{attribute addProperty BoxType "BK1250-0000-0019"}
{attribute addProperty Id "A_0001_KL_6211_ASI_Master_Parameter_Interface_and_6_Byte_11_ASI_Slaves_PowerKL6211_9210FF7200A_0002_KL_6211_ASI_Master_Parameter_Interface_and_6_Byte_11_ASI_Slaves_PowerKL_F309D72200A_0005_KL_6211_ASI_Master_Parameter_Interface_and_16_Byte_31_ASI_Slaves_PowerKL_54D8646000A_0006_KL_6211_ASI_Master_Parameter_Interface_and_16_Byte_31_ASI_Slaves_PowerKL_ACEFA9F000A_0009_KL_6211_ASI_Master_Parameter_Interface_and_32_Byte_62_ASI_Slaves_PowerKL_147C221C00A_0010_KL_6211_ASI_Master_Parameter_Interface_and_32_Byte_62_ASI_Slaves_PowerKL_6FFC768800A_0012_KL_6224_IO_Link_Master_Parameter_Interface_and_6_Byte_Process_DataKL6224_D683A81500A_0013_KL_6224_IO_Link_Master_Parameter_Interface_and_18_Byte_Process_DataKL_6B0FFD8100A_0014_KL_6224_IO_Link_Master_Parameter_Interface_and_30_Byte_Process_DataKL_D90EE1F900A_0015_KL_6224_IO_Link_Master_Parameter_Interface_and_42_Byte_Process_DataKL_C65F41F700A_0016_KL_6301_EIB_24_BYTE_InterfaceKL_D8C40AF800A_0017_KL_6401_LON_36_BYTE_InterfaceKL_614D78AA00A_0018_KM_6551_IEEE802_15_4_12_Byte_InterfaceKL6551_7AF854FD00A_0019_KL_6581_EnOcean_12_BYTE_InterfaceKL_F3D6C44700A_0020_KM_6663_Ethernet_Changeover_SwitchKL_4CCC064A00A_0021_KL_6771_MP_BUS_Master_12_Byte_InterfaceKL_7AF854FD00A_0022_KL_6781_M_Bus_Interface_22_ByteKL6781_3B6B34A300A_0023_KL_6811_DALI_Master_with_Power_SupplierKL6811_A76F47FB00A_0024_KL_6821_DALI_2_Multi_Master_with_Power_SupplierKL6821_3202269B00A_0025_KL_6831_SMI_LoVo_Interface_22_ByteKL6831_3B6B34A300A_0026_KL_6841_SMI_AC_Interface_22_ByteKL6841_3B6B34A300A_0027_KL_6904_Safety_Logic_7_TwinSAFE_ConnectionsKL6904_172C742100A_0028_KL_6904_Safety_Logic_15_TwinSAFE_ConnectionsKL_064A9C4500A_0029_KL_8001_Powerterminal_1ChKL_C24BBF3E00A_0030_KL_8001_Powerterminal_3_ChKL8001_77AB208D00A_0031_KL_8519_16_digital_InputKL8519_AEDCEC5800A_0032_KL_8524_2x4_digital_OutputKL8524_E623539600A_0033_KL_8528_8_digital_OutputKL8528_B5B8BA9000A_0034_KL_8548_8_Ch_ana_Output_0_10VKL8548_AC6A7E6D00A_0035_KL_8610_1_Ch_Adapter_KL8601KL8610_090A582100A_0036_KL_8610_2_Ch_Adapter_KL8601KL_4EE76BF900A_0037_KL_8610_3_Ch_Adapter_KL8601KL_F9570BBC00A_0038_KL_8610_4_Ch_Adapter_KL8601KL_8093826800A_0039_KL_8610_5_Ch_Adapter_KL8601KL_8108FB2E00A_0040_KL_8610_6_Ch_Adapter_KL8601KL_A3A627BC00A_0041_KL_8610_7_Ch_Adapter_KL8601KL_AF6F1E8600A_0042_KL_8610_8_Ch_Adapter_KL8601KL_57B9D98800A_0050_KL_9110_Power_Supplier_with_LED_and_Diag_24VKL9110_9CB5E82700A_0052_KL_9160_Power_Supplier_with_LED_and_Diag_230VKL9160_9CB5E82700A_0064_KL_9191_Dig_I_OKL9191_35652C4F00A_0067_KL_9210_Power_Supplier_with_Fuse_LED_and_Diag_24VKL9210_9CB5E82700A_0069_KL_9260_Power_Supplier_with_Fuse_LED_and_Diag_230VKL9260_9CB5E82700A_0078_KL_9505_0010_Power_Supplier_5V_0_5A_DiagKL_6FBA828600A_0080_KL_9508_0010_Power_Supplier_8V_0_5A_DiagKL_6FBA828600A_0082_KL_9510_0010_Power_Supplier_10V_0_5A_DiagKL_6FBA828600A_0084_KL_9512_0010_Power_Supplier_12V_0_5A_DiagKL_6FBA828600A_0086_KL_9515_0010_Power_Supplier_15V_0_5A_DiagKL_6FBA828600A_0087_KL_9528_Power_Supplier_AS_i_2AKL9528_5A9EA7C200A_0092_KLWORD_1_In_and_1_Output_WordKL9999_BA48D3D000"}
{attribute addProperty CRC "144214153"}
{attribute addProperty SizeInBites "0"}
{attribute addProperty SizeInBytes "0"}
TYPE TcTerminals210_2BK1250_08988889 EXTENDS BK1250_A5F67C82 :
STRUCT
	{attribute addProperty Name "A_0001_KL_6211_ASI_Master_Parameter_Interface_and_6_Byte_11_ASI_Slaves_Power"}
	A_0001_KL_6211_ASI_Master_Parameter_Interface_and_6_Byte_11_ASI_Slaves_Power : KL6211_9210FF72;
	{attribute addProperty Name "A_0002_KL_6211_ASI_Master_Parameter_Interface_and_6_Byte_11_ASI_Slaves_Power"}
	A_0002_KL_6211_ASI_Master_Parameter_Interface_and_6_Byte_11_ASI_Slaves_Power : KL_F309D722;
	{attribute addProperty Name "A_0005_KL_6211_ASI_Master_Parameter_Interface_and_16_Byte_31_ASI_Slaves_Power"}
	A_0005_KL_6211_ASI_Master_Parameter_Interface_and_16_Byte_31_ASI_Slaves_Power : KL_54D86460;
	{attribute addProperty Name "A_0006_KL_6211_ASI_Master_Parameter_Interface_and_16_Byte_31_ASI_Slaves_Power"}
	A_0006_KL_6211_ASI_Master_Parameter_Interface_and_16_Byte_31_ASI_Slaves_Power : KL_ACEFA9F0;
	{attribute addProperty Name "A_0009_KL_6211_ASI_Master_Parameter_Interface_and_32_Byte_62_ASI_Slaves_Power"}
	A_0009_KL_6211_ASI_Master_Parameter_Interface_and_32_Byte_62_ASI_Slaves_Power : KL_147C221C;
	{attribute addProperty Name "A_0010_KL_6211_ASI_Master_Parameter_Interface_and_32_Byte_62_ASI_Slaves_Power"}
	A_0010_KL_6211_ASI_Master_Parameter_Interface_and_32_Byte_62_ASI_Slaves_Power : KL_6FFC7688;
	{attribute addProperty Name "A_0012_KL_6224_IO_Link_Master_Parameter_Interface_and_6_Byte_Process_Data"}
	A_0012_KL_6224_IO_Link_Master_Parameter_Interface_and_6_Byte_Process_Data : KL6224_D683A815;
	{attribute addProperty Name "A_0013_KL_6224_IO_Link_Master_Parameter_Interface_and_18_Byte_Process_Data"}
	A_0013_KL_6224_IO_Link_Master_Parameter_Interface_and_18_Byte_Process_Data : KL_6B0FFD81;
	{attribute addProperty Name "A_0014_KL_6224_IO_Link_Master_Parameter_Interface_and_30_Byte_Process_Data"}
	A_0014_KL_6224_IO_Link_Master_Parameter_Interface_and_30_Byte_Process_Data : KL_D90EE1F9;
	{attribute addProperty Name "A_0015_KL_6224_IO_Link_Master_Parameter_Interface_and_42_Byte_Process_Data"}
	A_0015_KL_6224_IO_Link_Master_Parameter_Interface_and_42_Byte_Process_Data : KL_C65F41F7;
	{attribute addProperty Name "A_0016_KL_6301_EIB_24_BYTE_Interface"}
	A_0016_KL_6301_EIB_24_BYTE_Interface : KL_D8C40AF8;
	{attribute addProperty Name "A_0017_KL_6401_LON_36_BYTE_Interface"}
	A_0017_KL_6401_LON_36_BYTE_Interface : KL_614D78AA;
	{attribute addProperty Name "A_0018_KM_6551_IEEE802_15_4_12_Byte_Interface"}
	A_0018_KM_6551_IEEE802_15_4_12_Byte_Interface : KL6551_7AF854FD;
	{attribute addProperty Name "A_0019_KL_6581_EnOcean_12_BYTE_Interface"}
	A_0019_KL_6581_EnOcean_12_BYTE_Interface : KL_F3D6C447;
	{attribute addProperty Name "A_0020_KM_6663_Ethernet_Changeover_Switch"}
	A_0020_KM_6663_Ethernet_Changeover_Switch : KL_4CCC064A;
	{attribute addProperty Name "A_0021_KL_6771_MP_BUS_Master_12_Byte_Interface"}
	A_0021_KL_6771_MP_BUS_Master_12_Byte_Interface : KL_7AF854FD;
	{attribute addProperty Name "A_0022_KL_6781_M_Bus_Interface_22_Byte"}
	A_0022_KL_6781_M_Bus_Interface_22_Byte : KL6781_3B6B34A3;
	{attribute addProperty Name "A_0023_KL_6811_DALI_Master_with_Power_Supplier"}
	A_0023_KL_6811_DALI_Master_with_Power_Supplier : KL6811_A76F47FB;
	{attribute addProperty Name "A_0024_KL_6821_DALI_2_Multi_Master_with_Power_Supplier"}
	A_0024_KL_6821_DALI_2_Multi_Master_with_Power_Supplier : KL6821_3202269B;
	{attribute addProperty Name "A_0025_KL_6831_SMI_LoVo_Interface_22_Byte"}
	A_0025_KL_6831_SMI_LoVo_Interface_22_Byte : KL6831_3B6B34A3;
	{attribute addProperty Name "A_0026_KL_6841_SMI_AC_Interface_22_Byte"}
	A_0026_KL_6841_SMI_AC_Interface_22_Byte : KL6841_3B6B34A3;
	{attribute addProperty Name "A_0027_KL_6904_Safety_Logic_7_TwinSAFE_Connections"}
	A_0027_KL_6904_Safety_Logic_7_TwinSAFE_Connections : KL6904_172C7421;
	{attribute addProperty Name "A_0028_KL_6904_Safety_Logic_15_TwinSAFE_Connections"}
	A_0028_KL_6904_Safety_Logic_15_TwinSAFE_Connections : KL_064A9C45;
	{attribute addProperty Name "A_0029_KL_8001_Powerterminal_1Ch"}
	A_0029_KL_8001_Powerterminal_1Ch : KL_C24BBF3E;
	{attribute addProperty Name "A_0030_KL_8001_Powerterminal_3_Ch"}
	A_0030_KL_8001_Powerterminal_3_Ch : KL8001_77AB208D;
	{attribute addProperty Name "A_0031_KL_8519_16_digital_Input"}
	A_0031_KL_8519_16_digital_Input : KL8519_AEDCEC58;
	{attribute addProperty Name "A_0032_KL_8524_2x4_digital_Output"}
	A_0032_KL_8524_2x4_digital_Output : KL8524_E6235396;
	{attribute addProperty Name "A_0033_KL_8528_8_digital_Output"}
	A_0033_KL_8528_8_digital_Output : KL8528_B5B8BA90;
	{attribute addProperty Name "A_0034_KL_8548_8_Ch_ana_Output_0_10V"}
	A_0034_KL_8548_8_Ch_ana_Output_0_10V : KL8548_AC6A7E6D;
	{attribute addProperty Name "A_0035_KL_8610_1_Ch_Adapter_KL8601"}
	A_0035_KL_8610_1_Ch_Adapter_KL8601 : KL8610_090A5821;
	{attribute addProperty Name "A_0036_KL_8610_2_Ch_Adapter_KL8601"}
	A_0036_KL_8610_2_Ch_Adapter_KL8601 : KL_4EE76BF9;
	{attribute addProperty Name "A_0037_KL_8610_3_Ch_Adapter_KL8601"}
	A_0037_KL_8610_3_Ch_Adapter_KL8601 : KL_F9570BBC;
	{attribute addProperty Name "A_0038_KL_8610_4_Ch_Adapter_KL8601"}
	A_0038_KL_8610_4_Ch_Adapter_KL8601 : KL_80938268;
	{attribute addProperty Name "A_0039_KL_8610_5_Ch_Adapter_KL8601"}
	A_0039_KL_8610_5_Ch_Adapter_KL8601 : KL_8108FB2E;
	{attribute addProperty Name "A_0040_KL_8610_6_Ch_Adapter_KL8601"}
	A_0040_KL_8610_6_Ch_Adapter_KL8601 : KL_A3A627BC;
	{attribute addProperty Name "A_0041_KL_8610_7_Ch_Adapter_KL8601"}
	A_0041_KL_8610_7_Ch_Adapter_KL8601 : KL_AF6F1E86;
	{attribute addProperty Name "A_0042_KL_8610_8_Ch_Adapter_KL8601"}
	A_0042_KL_8610_8_Ch_Adapter_KL8601 : KL_57B9D988;
	{attribute addProperty Name "A_0050_KL_9110_Power_Supplier_with_LED_and_Diag_24V"}
	A_0050_KL_9110_Power_Supplier_with_LED_and_Diag_24V : KL9110_9CB5E827;
	{attribute addProperty Name "A_0052_KL_9160_Power_Supplier_with_LED_and_Diag_230V"}
	A_0052_KL_9160_Power_Supplier_with_LED_and_Diag_230V : KL9160_9CB5E827;
	{attribute addProperty Name "A_0064_KL_9191_Dig_I_O"}
	A_0064_KL_9191_Dig_I_O : KL9191_35652C4F;
	{attribute addProperty Name "A_0067_KL_9210_Power_Supplier_with_Fuse_LED_and_Diag_24V"}
	A_0067_KL_9210_Power_Supplier_with_Fuse_LED_and_Diag_24V : KL9210_9CB5E827;
	{attribute addProperty Name "A_0069_KL_9260_Power_Supplier_with_Fuse_LED_and_Diag_230V"}
	A_0069_KL_9260_Power_Supplier_with_Fuse_LED_and_Diag_230V : KL9260_9CB5E827;
	{attribute addProperty Name "A_0078_KL_9505_0010_Power_Supplier_5V_0_5A_Diag"}
	A_0078_KL_9505_0010_Power_Supplier_5V_0_5A_Diag : KL_6FBA8286;
	{attribute addProperty Name "A_0080_KL_9508_0010_Power_Supplier_8V_0_5A_Diag"}
	A_0080_KL_9508_0010_Power_Supplier_8V_0_5A_Diag : KL_6FBA8286;
	{attribute addProperty Name "A_0082_KL_9510_0010_Power_Supplier_10V_0_5A_Diag"}
	A_0082_KL_9510_0010_Power_Supplier_10V_0_5A_Diag : KL_6FBA8286;
	{attribute addProperty Name "A_0084_KL_9512_0010_Power_Supplier_12V_0_5A_Diag"}
	A_0084_KL_9512_0010_Power_Supplier_12V_0_5A_Diag : KL_6FBA8286;
	{attribute addProperty Name "A_0086_KL_9515_0010_Power_Supplier_15V_0_5A_Diag"}
	A_0086_KL_9515_0010_Power_Supplier_15V_0_5A_Diag : KL_6FBA8286;
	{attribute addProperty Name "A_0087_KL_9528_Power_Supplier_AS_i_2A"}
	A_0087_KL_9528_Power_Supplier_AS_i_2A : KL9528_5A9EA7C2;
	{attribute addProperty Name "A_0092_KLWORD_1_In_and_1_Output_Word"}
	A_0092_KLWORD_1_In_and_1_Output_Word : KL9999_BA48D3D0;
END_STRUCT
END_TYPE

(* stored: Version 1.2.0.0, ProductVersion 3.1.4024.9
   DUT TcTerminals210_2BK1250_08988889: Id {d6761338-ceec-444f-8d81-9d61d537d592} *)
